(*
  QualiVision line camera system
  DMAX76.   
*)
FUNCTION_BLOCK FB_LineCamera76 EXTENDS FB_LineCamera

VAR CONSTANT
  cCameraWidth76            : DINT :=  9216;   (*Camera width [px]*)
  cCameraMechOffsetTC76     : REAL := 101.5;   (*Camera mechanical offset at calibration temp [mm]*)
  cMechOffsetCameraToPU76   : REAL :=  13.039; (*Camera mechanical offset to PrintUnit [mm]*)
  cPrintUnitMechOffsetTC76  : REAL := 32.9869; (*PrintUnit mechanical offset at calibration temp [mm]*)
END_VAR

SUPER^();

METHOD InitLineCamera
VAR_INPUT
  nPrintUnitResolution         : UDINT;    (*printhead pixel resolution [dpi]*)
  nPrintUnitSubPx              : UDINT;    (*print unit subPixel resolution [SubPx]*)
  nPrintUnitWidth              : UDINT;    (*print unit width in [px]*)
  iCameraTrigger               : I_CameraTrigger;
END_VAR
(*Init for dmax type*)
_nCameraWidth           := cCameraWidth76;
_fCameraMechOffsetTC    := cCameraMechOffsetTC76;
_fMechOffsetCameraToPU  := cMechOffsetCameraToPU76;
_fPrintUnitMechOffsetTC := cPrintUnitMechOffsetTC76;

SUPER^.InitLineCamera( nPrintUnitResolution := nPrintUnitResolution
                      , nPrintUnitSubPx := nPrintUnitSubPx
                      , nPrintUnitWidth := nPrintUnitWidth
                      , iCameraTrigger := iCameraTrigger);
END_METHOD

{attribute 'monitoring':='variable'}
PROPERTY sName : STRING
GET
sName := 'LineCam 76';
END_GET
END_PROPERTY

END_FUNCTION_BLOCK

(* stored: Version 1.1.0.1, ProductVersion 3.1.4024.3
   POU FB_LineCamera76: Id {15ceca3a-7103-4457-a274-7252f0c4f78a}, SpecialFunc None
   Method InitLineCamera: Id {e06e6bbe-fd53-41c2-a6db-688c998f8313}
   Property sName: Id {8301cae9-7d38-4a93-89ac-c559b839d964}
   Get Get: Id {85e4ef51-1389-464c-b3b5-e990c62c96db} *)
